FUNCTION_BLOCK PUBLIC ProductionPlaner EXTENDS TcoCore.TcoRemoteTask
VAR_INPUT
END_VAR
VAR_OUTPUT
END_VAR
VAR
	_productonPlanCompleted: BOOL;
	_productionPlanIsEmpty: BOOL;
	_requiredProcessSettings: STRING;
END_VAR

super^();

PROPERTY PUBLIC ProductionPlanCompleted : bool
GET
ProductionPlanCompleted:=_productonPlanCompleted;
END_GET
END_PROPERTY

PROPERTY PUBLIC ProductionPlanIsEmpty : bool
GET
ProductionPlanIsEmpty:=_productionPlanIsEmpty;
END_GET
END_PROPERTY

PROPERTY RequiredProcessSettingsId : string
GET
RequiredProcessSettingsId:=_requiredProcessSettings;
END_GET
END_PROPERTY

(*~
	<docu>
		<summary>
			Restores this instance to the Ready state. Can be called explicitly or from within one of the restore mechanisms.
			<para>
				See also <see cref="PlcDocu.TcoCore.TcoTask.AutoRestorable()"/>
			</para>
		</summary>			
	</docu>	
~*)
METHOD Restore : ITcoRestorable
SUPER^.Restore();
_productonPlanCompleted:=FALSE;
_productionPlanIsEmpty:=FALSE;
_requiredProcessSettings:='';
END_METHOD

END_FUNCTION_BLOCK

(* stored: Version 1.1.0.1
   POU ProductionPlaner: Id {8e167958-6b6e-4b49-a6ec-53d5acd89358}, SpecialFunc None
   Property ProductionPlanCompleted: Id {2b0a59d7-c9ae-4b8b-b474-b91a4ce77769}
   Get Get: Id {52a1820b-f039-4cce-b8e5-65a5c21fe408}
   Property ProductionPlanIsEmpty: Id {fabb3d56-595f-45a4-a452-c9ee378a14c5}
   Get Get: Id {b532c513-17bd-48a3-97ed-ee0f5c9ebffc}
   Property RequiredProcessSettingsId: Id {cca1091f-75a0-427f-8ffb-c2ac68f7dabe}
   Get Get: Id {0875d524-7597-4c79-84e1-47a84b2def08}
   Method Restore: Id {3fbf695e-6100-468e-8bd4-f042b4c127b6} *)
